PROGRAM EncoderMeas
VAR
	
encoder1:ENCODERPULSEtoANGLE;

END_VAR

//Dónde estoy?
///Medir ángulos
encoder1.A:=IO.encoder1_A;
encoder1.B:=IO.encoder1_B;
encoder1();
GVL.alfa:=encoder1.angle;

END_PROGRAM

(* stored: Version 1.1.0.1, ProductVersion 3.1.4024.4
   POU EncoderMeas: Id {0d96bc1c-ffb1-440d-b63c-eed900a16197}, SpecialFunc None *)
